GLOBALCONSTANTS DefaultPool_TC_SC (* Global constants *)
  PACKAGE Uebungen::const::UT::TC_SC;
  VAR_GLOBAL CONSTANT
    ISO_DESIGNATOR_WIDTH : UINT := 160;
    ISO_DESIGNATOR_HEIGHT : UINT := 80;
    ISO_MASK_SIZE : UINT := 480;
    ISO_VERSION_LABEL : STRING;
    MASK_WIDTH : UINT := 480;
    MASK_HEIGHT : UINT := 480;
    WorkingSet : UINT := 0;
    DataMask : UINT := 1000;
    OutputString_TC_SC : UINT := 11500;
    FontAttributes_SKM : UINT := 23500;
  END_VAR
END_GLOBALCONSTANTS
